{attribute addProperty BoxType "EL3483-0060-0018"}
{attribute addProperty Id "VoltageAT %I*REAL324"}
{attribute addProperty CRC "4266836333"}
{attribute addProperty SizeInBites "32"}
{attribute addProperty SizeInBytes "4"}
TYPE L2_Basic_FE52C16D :
STRUCT
	{attribute addProperty Name "Voltage"}
	Voltage AT %I* : REAL;
END_STRUCT
END_TYPE

(* stored: Version 1.2.0.0, ProductVersion 3.1.4024.9
   DUT L2_Basic_FE52C16D: Id {105e8c3b-647c-4704-b829-421d96a150fa} *)
